Universal Robots PolyScope program: testing.urp

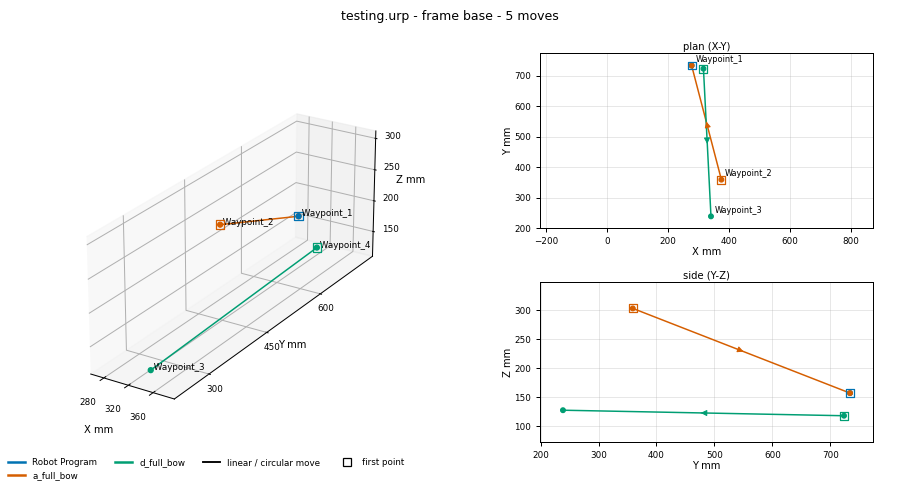
[picture p0: tool path of testing.urp in frame base, 5 of 6 moves have a stored position in this frame; points joined in program order, loops and branches not executed]
Program testing (installation=string_planes directory=/programs createdIn=5.17.3 lastSavedIn=5.17.3 robotSerialNumber=20245501435)
Calibrated DH parameters: a=[0.000154, -0.137004, -0.385524, -0.00002, 0.000092, 0]; d=[0.162441, 211.794786, -230.585024, 18.923638, 0.099786, 0.09951]; alpha=[1.569493, -0.001902, 0.003874, 1.570111, -1.570167, 0]; deltaTheta=[0, -1.242934, 1.056292, 0.186646, 0.000002, 0.000001]
InitVariablesNode
Robot Program (runOnlyOnce=false)
  MoveJ speed 60 deg/s, acceleration 80 deg/s^2 (useActiveTCP=true) feature=Base
    Waypoint Waypoint_1: TCP in base x=277.237 y=734.032 z=156.892 mm, rx=1.7389 ry=2.3104 rz=-1.1078 rad; joints [-126.647, -28.123, 54.729, -74.616, -91.964, -141.812] deg; TCP offset x=28.21 y=-96.107 z=-99.69 mm, rx=0 ry=0 rz=0 rad
  bow_dir := True
  note_dur := 1
  Call a_full_bow
  Call a_to_d
  bow_dir := False
  Call d_full_bow
  Halt
SubProgram -> d_full_bow
SubProgram -> a_to_d
SubProgram -> a_full_bow
SubProgram a_full_bow (keepSynchronizedWithDisk=false) programFile=/programs/a_full_bow.urp
  Timer (action=Start) variable(name=timer_1)
  If bow_dir
    MoveL speed 250 mm/s, acceleration 1200 mm/s^2 (useActiveTCP=true) feature=Base
      Waypoint Waypoint_2: TCP in base x=374.969 y=359.127 z=303.035 mm, rx=1.6275 ry=2.3373 rz=-1.1146 rad; joints [-156.117, -66.368, 101.552, -88.734, -114.429, -168.118] deg; TCP offset x=28.21 y=-96.107 z=-99.69 mm, rx=0 ry=0 rz=0 rad
        Until EXPRESSION (allowActions=false) ExpressionBranch=timer_1≟note_dur
  Else 
    MoveL speed 250 mm/s, acceleration 1200 mm/s^2 (useActiveTCP=true) feature=Base
      Waypoint Waypoint_1: TCP in base x=277.237 y=734.032 z=156.892 mm, rx=1.7389 ry=2.3104 rz=-1.1078 rad; joints [-126.647, -28.123, 54.729, -74.616, -91.964, -141.812] deg; TCP offset x=28.21 y=-96.107 z=-99.69 mm, rx=0 ry=0 rz=0 rad
        Until EXPRESSION (allowActions=false) ExpressionBranch=timer_1≟note_dur
  SuppressedNode
    MoveL speed 250 mm/s, acceleration 1200 mm/s^2 (useActiveTCP=true) feature=Base
      Waypoint Waypoint_1: TCP in base x=277.237 y=734.032 z=156.892 mm, rx=1.7389 ry=2.3104 rz=-1.1078 rad; joints [-126.647, -28.123, 54.729, -74.616, -91.964, -141.812] deg
      Waypoint Waypoint_3: motionParameters(blendRadius=0.05); TCP in base x=335.809 y=527.638 z=230.762 mm, rx=1.7389 ry=2.3104 rz=-1.1078 rad; joints [-141.244, -51.172, 87.867, -86.053, -101.589, -152.842] deg; TCP offset x=28.21 y=-96.107 z=-99.69 mm, rx=0 ry=0 rz=0 rad
      Waypoint Waypoint_2: TCP in base x=393.128 y=325.659 z=303.053 mm, rx=1.7389 ry=2.3104 rz=-1.1078 rad; joints [-160.523, -67.347, 103.242, -90.17, -113.569, -168.748] deg
  Timer (action=Stop) variable=timer_1
  Timer (action=Reset) variable=timer_1
SubProgram a_to_d (keepSynchronizedWithDisk=false) programFile=/programs/a_to_d.urp
  MoveJ speed 60 deg/s, acceleration 80 deg/s^2 (useActiveTCP=true) feature=Base
    Waypoint Waypoint_9 (Relative): relativeFromPosition TCP in base x=327.369 y=541.717 z=231.872 mm, rx=1.6817 ry=2.3248 rz=-1.1114 rad; joints [-139.639, -50.321, 85.997, -84.695, -102.359, -153.08] deg; TCP in base x=337.287 y=452.573 z=146.265 mm, rx=-1.6084 ry=-2.1977 rz=1.0429 rad; joints [-146.228, -47.168, 100.748, -99.802, -91.44, -163.024] deg
SubProgram d_full_bow (keepSynchronizedWithDisk=false) programFile=/programs/d_full_bow.urp
  Timer (action=Start) variable=timer_1
  If bow_dir≟ False
    MoveL speed 250 mm/s, acceleration 1200 mm/s^2 (useActiveTCP=true) feature=Base
      Waypoint Waypoint_4: TCP in base x=316.077 y=723.624 z=117.8 mm, rx=-1.5349 ry=-2.2386 rz=1.1274 rad; joints [-128.458, -21.868, 50.818, -72.931, -81.953, -152.853] deg
        Until EXPRESSION (allowActions=false) ExpressionBranch=timer_1≟note_dur
  Else 
    MoveL speed 250 mm/s, acceleration 1200 mm/s^2 (useActiveTCP=true) feature=Base
      Waypoint Waypoint_3: TCP in base x=340.806 y=238.625 z=127.338 mm, rx=-1.5375 ry=-2.1223 rz=1.0863 rad; joints [-167.854, -53.469, 123.568, -113.681, -104.543, -179.466] deg
        Until EXPRESSION (allowActions=false) ExpressionBranch=timer_1≟note_dur
  SuppressedNode
    MoveL speed 250 mm/s, acceleration 1200 mm/s^2 (useActiveTCP=true) feature=Base
      Waypoint Waypoint_1: TCP in base x=331.973 y=720.894 z=108.291 mm, rx=-1.645 ry=-2.1081 rz=1.0591 rad; joints [-129.773, -21.651, 52.373, -76.468, -76.907, -149.022] deg
      Waypoint Waypoint_2: motionParameters(blendRadius=0.05); TCP in base x=332.259 y=481.199 z=108.291 mm, rx=-1.645 ry=-2.1081 rz=1.0591 rad; joints [-144.031, -41.816, 97.865, -100.392, -86.961, -159.136] deg
      Waypoint Waypoint_3: TCP in base x=332.566 y=223.853 z=108.291 mm, rx=-1.645 ry=-2.1081 rz=1.0591 rad; joints [-170.229, -51.627, 126.122, -120.942, -105.516, -177.767] deg
  Timer (action=Stop) variable=timer_1
  Timer (action=Reset) variable=timer_1
